{region '#Template'}
	{attribute 'Version' := '1.0.0.0'}
	{attribute 'Tags' := '"LCID": "1031", "Text": "H, General, HtgCir, Operating mode"'}
	{attribute 'Tags' := '"LCID": "1033", "Text": "H, General, HtgCir, Operating mode"'}
	{attribute 'Description' := '"LCID": "1031", "Text": "Heizgrenzwert"'}
	{attribute 'Description' := '"LCID": "1033", "Text": "Heating limit"'}
{endregion}
FUNCTION_BLOCK FB_BA_HtgLmt EXTENDS FB_BA_View
VAR_INPUT
	fIn						: REAL;
END_VAR
VAR_OUTPUT
	bQ						: BOOL;
END_VAR
VAR_INPUT CONSTANT
	Sp						: FB_BA_AV_Op;	
	Q						: FB_BA_BV_Op;		
END_VAR	
VAR
	Swi2P					: FB_BA_Swi2P;
END_VAR
VAR // added by the converter: edge detectors and wires of the graphical bodies
    _w1 : ANY;
END_VAR

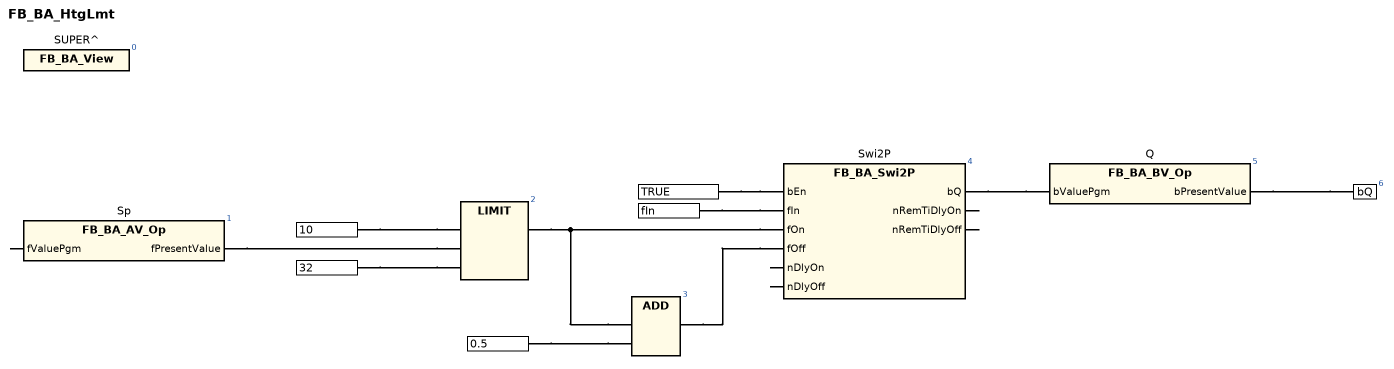
SUPER^(); // FB_BA_View
Sp(); // FB_BA_AV_Op
_w1 := LIMIT(10, Sp.fPresentValue, 32);
Swi2P(bEn := TRUE, fIn := fIn, fOn := _w1, fOff := _w1 + 0.5); // FB_BA_Swi2P
Q(bValuePgm := Swi2P.bQ); // FB_BA_BV_Op
bQ := Q.bPresentValue;

METHOD FB_init : BOOL
VAR_INPUT
	bInitRetains : BOOL; // if TRUE, the retain variables are initialized (warm start / cold start)
	bInCopyCode : BOOL;  // if TRUE, the instance afterwards gets moved into the copy code (online change)
END_VAR
Sp.iParent			:= THIS^;
Sp.iLabel			:= LblCmpHeating.HtgLmt_Sp;
Sp.sObjectName		:= '{Idx=01}';								 	 
Sp.eUnit			:= E_BA_Unit.eTemperature_DegreesCelsius;  
Sp.fValueRm			:= 16.0;
Sp.fCOVIncrement	:= BA2_Param.fDefCOVIncrement;							

Q.iParent			:= THIS^;
Q.iLabel			:= LblCmpHeating.HtgLmt_Q;												 
Q.sObjectName		:= '{Idx=01}';
Q.sActiveText		:= txtEvent_On;
Q.sInactiveText		:= txtEvent_Off;
Q.bValueRm			:= FALSE;								
Q.eToggleMode 		:= E_BA_ToggleMode.eSwitch;
END_METHOD

END_FUNCTION_BLOCK

(* stored: Version 1.1.0.1, ProductVersion 3.1.4024.9
   POU FB_BA_HtgLmt: Id {4e6f22bd-6796-4198-8ef8-b62c27af77c9}, SpecialFunc None
   Method FB_init: Id {b75e13ed-7d1d-4f1d-a86f-297276910a13} *)
